// TIA Portal V21 export
TYPE "Std_Paratia"
   STRUCT
      In : Struct
         SetpointAuto : Real;
         PulsanteIncrementa : Bool;
         PulsanteDecrementa : Bool;
         TermicoIntervenuto : Bool;
         FinecorsaPositivo : Bool;
         FinecorsaNegativo : Bool;
         AbilitazioneMovimento : Bool;
      END_STRUCT;
      Prm : Struct
         IsteresiComando : Real;
         UnitaMisura : "Std_UnitàDiMisura";
         AbilitazioneInterpolazione { S7_SetPoint := 'True'} : Bool := False;
         Interpolazione : Array[0..5] of Struct
            Setpoint : Real;
            Valore : Real;
         END_STRUCT;
      END_STRUCT;
      Dati : Struct
         AnalogicaReale : Real;
         PosizioneAttuale : Real;
         IncrementaUscita : Bool;
         PosizionePrecedente : Real;
         DeltaMovimentoTotale { S7_SetPoint := 'True'} : Real;
         DeltaMovimentoTotalePrecedente : Real;
         VerificaOvertime : Bool;
         InAllarme : Bool;
         ForzataChiusa : Bool;   // La paratia viene chiusa da condizioni esterne
      END_STRUCT;
      Hmi : Struct
         Auto : Bool;
         Man : Bool;
         PulsanteIncrementa : Bool;
         PulsanteDecrementa : Bool;
         Simulazione : Bool;
         SetpointBloccato : Bool;
      END_STRUCT;
      Allarmi : Struct
         TimerRitMov : "Std_stTimer";
         PresetSoglie : Struct
            MinimoSpostamento : Real;
         END_STRUCT;
         "A" : Array[0.."K_NumAllarmiPerParatie"] of "Std_PrmAllarmeStd";
         WordHMI : Word;
      END_STRUCT;
      Out : Struct
         CmdPos : Bool;
         CmdNeg : Bool;
      END_STRUCT;
      Rif_Inc : Struct
         K_AnalogicaPosAttuale : Int;   // indica la posizione attuale della paratia
         K_AnalogicaRiferimento : Int;   // Indica le soglie che vengono utilizzate dalla paratia
         K_StazioneRiferimento : Int;
      END_STRUCT;
   END_STRUCT;
   // Prm.Interpolazione[0].Setpoint := 0.0;
   // Prm.Interpolazione[1].Setpoint := 20.0;
   // Prm.Interpolazione[2].Setpoint := 40.0;
   // Prm.Interpolazione[3].Setpoint := 60.0;
   // Prm.Interpolazione[4].Setpoint := 80.0;
   // Prm.Interpolazione[5].Setpoint := 100.0;
   // Prm.Interpolazione[0].Valore := 0.0;
   // Prm.Interpolazione[1].Valore := 20.0;
   // Prm.Interpolazione[2].Valore := 40.0;
   // Prm.Interpolazione[3].Valore := 60.0;
   // Prm.Interpolazione[4].Valore := 80.0;
   // Prm.Interpolazione[5].Valore := 100.0;
   // // Allarmi."A"[1] : Overtime di movimento
   // // Allarmi."A"[2] : Termico intervenuto
   // // Allarmi."A"[3] : Sezionatore aperto
END_TYPE
